% RSLogix 500 project I2P JOB 23 - ANDREW_HOEMMEN_BAK067.RSS, saved by version 10.00.00.00 %
PROJECT "ML03A"    % processor: Bul.1763 MicroLogix 1100 Series B %

PROGRAM FILES
  LAD 2   17 rungs

DATA FILES
  O0 OUTPUT  4 elements
  I1 INPUT  6 elements
  S2 STATUS  66 elements
  B3 BINARY  1 elements
  T4 TIMER  1 elements
  C5 COUNTER  2 elements
  R6 CONTROL  1 elements
  N7 INTEGER  1 elements
  F8 FLOAT  1 elements

LADDER 2
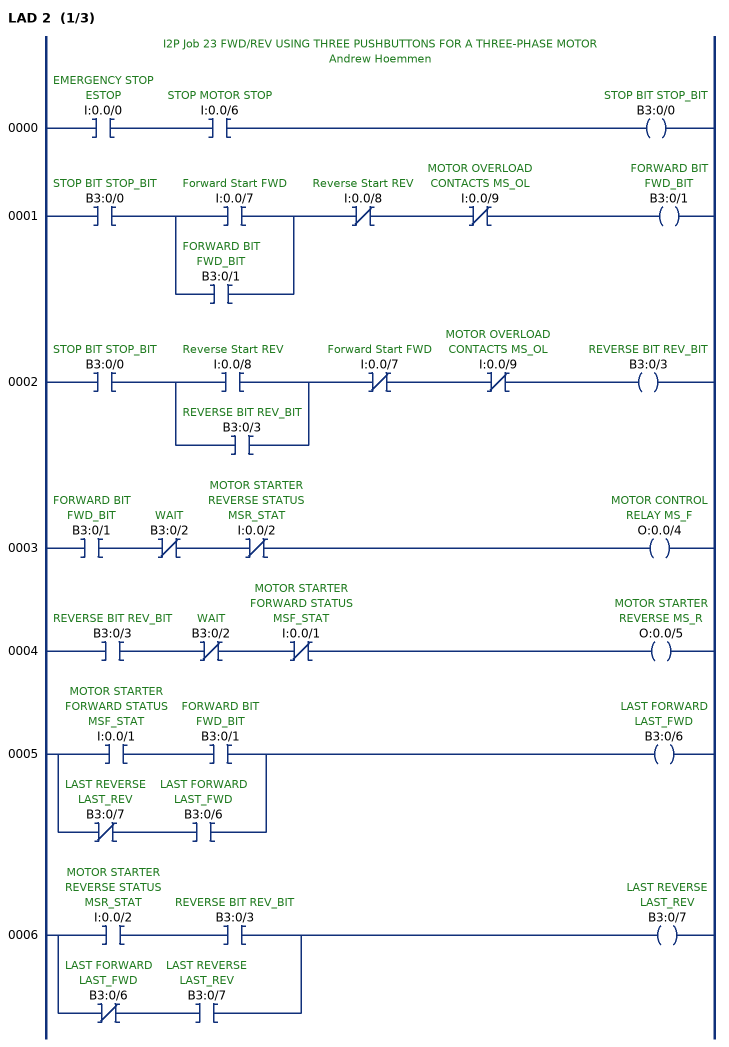
% Rung: 0 %
% I2P Job 23 FWD/REV USING THREE PUSHBUTTONS FOR A THREE-PHASE MOTOR
% Andrew Hoemmen %
SOR XIC I:0.0/0 XIC I:0.0/6 OTE B3:0/0 EOR
%   I:0.0/0  ESTOP  "EMERGENCY STOP" %
%   I:0.0/6  STOP  "STOP MOTOR" %
%   B3:0/0  STOP_BIT  "STOP BIT" %
% Rung: 1 %
SOR XIC B3:0/0 BST XIC I:0.0/7 NXB XIC B3:0/1 BND XIO I:0.0/8 XIO I:0.0/9 OTE B3:0/1 EOR
%   B3:0/0  STOP_BIT  "STOP BIT" %
%   I:0.0/7  FWD  "Forward Start" %
%   B3:0/1  FWD_BIT  "FORWARD BIT" %
%   I:0.0/8  REV  "Reverse Start" %
%   I:0.0/9  MS_OL  "MOTOR OVERLOAD CONTACTS" %
% Rung: 2 %
SOR XIC B3:0/0 BST XIC I:0.0/8 NXB XIC B3:0/3 BND XIO I:0.0/7 XIO I:0.0/9 OTE B3:0/3 EOR
%   B3:0/0  STOP_BIT  "STOP BIT" %
%   I:0.0/8  REV  "Reverse Start" %
%   B3:0/3  REV_BIT  "REVERSE BIT" %
%   I:0.0/7  FWD  "Forward Start" %
%   I:0.0/9  MS_OL  "MOTOR OVERLOAD CONTACTS" %
% Rung: 3 %
SOR XIC B3:0/1 XIO B3:0/2 XIO I:0.0/2 OTE O:0.0/4 EOR
%   B3:0/1  FWD_BIT  "FORWARD BIT" %
%   B3:0/2  WAIT %
%   I:0.0/2  MSR_STAT  "MOTOR STARTER REVERSE STATUS" %
%   O:0.0/4  MS_F  "MOTOR CONTROL RELAY" %
% Rung: 4 %
SOR XIC B3:0/3 XIO B3:0/2 XIO I:0.0/1 OTE O:0.0/5 EOR
%   B3:0/3  REV_BIT  "REVERSE BIT" %
%   B3:0/2  WAIT %
%   I:0.0/1  MSF_STAT  "MOTOR STARTER FORWARD STATUS" %
%   O:0.0/5  MS_R  "MOTOR STARTER REVERSE" %
% Rung: 5 %
SOR BST XIC I:0.0/1 XIC B3:0/1 NXB XIO B3:0/7 XIC B3:0/6 BND OTE B3:0/6 EOR
%   I:0.0/1  MSF_STAT  "MOTOR STARTER FORWARD STATUS" %
%   B3:0/1  FWD_BIT  "FORWARD BIT" %
%   B3:0/7  LAST_REV  "LAST REVERSE" %
%   B3:0/6  LAST_FWD  "LAST FORWARD" %
% Rung: 6 %
SOR BST XIC I:0.0/2 XIC B3:0/3 NXB XIO B3:0/6 XIC B3:0/7 BND OTE B3:0/7 EOR
%   I:0.0/2  MSR_STAT  "MOTOR STARTER REVERSE STATUS" %
%   B3:0/3  REV_BIT  "REVERSE BIT" %
%   B3:0/6  LAST_FWD  "LAST FORWARD" %
%   B3:0/7  LAST_REV  "LAST REVERSE" %

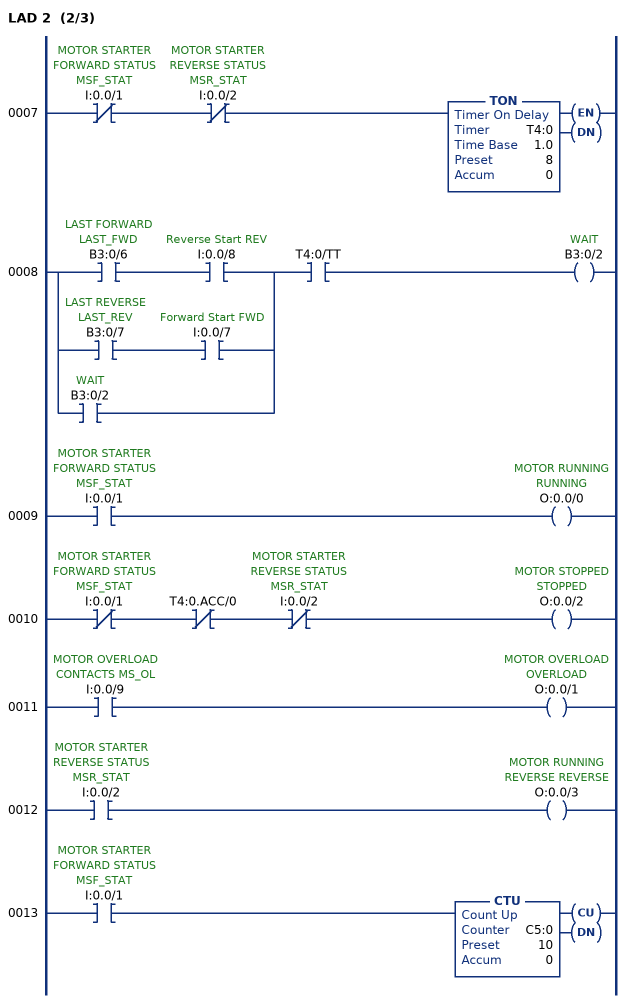
% Rung: 7 %
SOR XIO I:0.0/1 XIO I:0.0/2 TON T4:0 1.0 8 0 EOR
%   I:0.0/1  MSF_STAT  "MOTOR STARTER FORWARD STATUS" %
%   I:0.0/2  MSR_STAT  "MOTOR STARTER REVERSE STATUS" %
% Rung: 8 %
SOR BST XIC B3:0/6 XIC I:0.0/8 NXB BST XIC B3:0/7 XIC I:0.0/7 NXB XIC B3:0/2 BND BND XIC T4:0/TT OTE B3:0/2 EOR
%   B3:0/6  LAST_FWD  "LAST FORWARD" %
%   I:0.0/8  REV  "Reverse Start" %
%   B3:0/7  LAST_REV  "LAST REVERSE" %
%   I:0.0/7  FWD  "Forward Start" %
%   B3:0/2  WAIT %
% Rung: 9 %
SOR XIC I:0.0/1 OTE O:0.0/0 EOR
%   I:0.0/1  MSF_STAT  "MOTOR STARTER FORWARD STATUS" %
%   O:0.0/0  RUNNING  "MOTOR RUNNING" %
% Rung: 10 %
SOR XIO I:0.0/1 XIO T4:0.ACC/0 XIO I:0.0/2 OTE O:0.0/2 EOR
%   I:0.0/1  MSF_STAT  "MOTOR STARTER FORWARD STATUS" %
%   I:0.0/2  MSR_STAT  "MOTOR STARTER REVERSE STATUS" %
%   O:0.0/2  STOPPED  "MOTOR STOPPED" %
% Rung: 11 %
SOR XIC I:0.0/9 OTE O:0.0/1 EOR
%   I:0.0/9  MS_OL  "MOTOR OVERLOAD CONTACTS" %
%   O:0.0/1  OVERLOAD  "MOTOR OVERLOAD" %
% Rung: 12 %
SOR XIC I:0.0/2 OTE O:0.0/3 EOR
%   I:0.0/2  MSR_STAT  "MOTOR STARTER REVERSE STATUS" %
%   O:0.0/3  REVERSE  "MOTOR RUNNING REVERSE" %
% Rung: 13 %
SOR XIC I:0.0/1 CTU C5:0 10 0 EOR
%   I:0.0/1  MSF_STAT  "MOTOR STARTER FORWARD STATUS" %

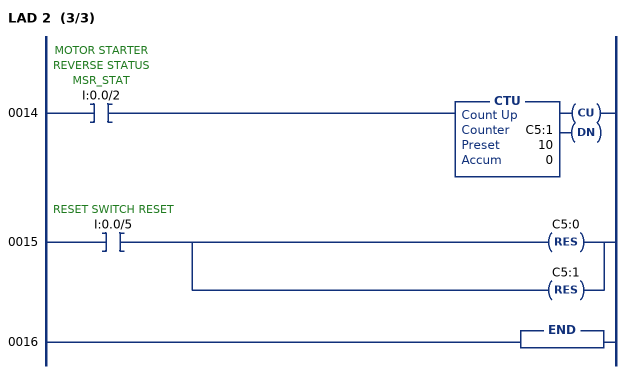
% Rung: 14 %
SOR XIC I:0.0/2 CTU C5:1 10 0 EOR
%   I:0.0/2  MSR_STAT  "MOTOR STARTER REVERSE STATUS" %
% Rung: 15 %
SOR XIC I:0.0/5 BST RES C5:0 NXB RES C5:1 BND EOR
%   I:0.0/5  RESET  "RESET SWITCH" %
% Rung: 16 %
SOR END EOR

OTHER DOCUMENTED ADDRESSES
  B3:0/4  REV_JOG  "REVERSE JOG"
  B3:0/5  CHAN_BIT  "CHANGING BIT"
  DIR_STATS  
  I:0.0/3  "MODE ON/OFF AUTO"
  I:0.0/4  MODE_ON  "MODE ON/OFF AUTO"
  T4:0.ACC  BLINK  "LIGHT BLINKING"

DATA TABLE (non-zero values as saved)
DATA T4
% .PRE .ACC %
% T4:0 % 8 0
DATA C5
% .PRE .ACC %
% C5:0 % 10 0
% C5:1 % 10 0
